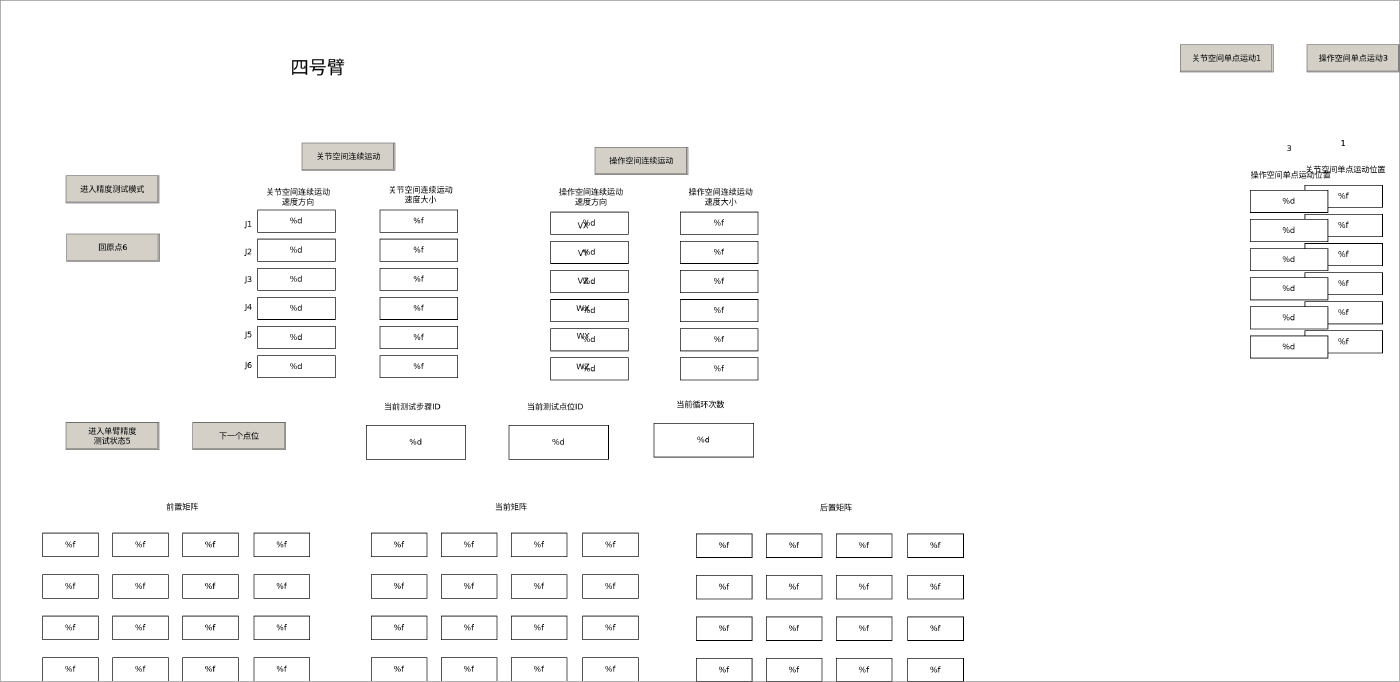
VISUALIZATION Robot_Jog_Arm4  // 1921x937
    Button (90,241 128x38), "进入精度测试模式", colour toggle: GVL_AccuracyTestVar.g_enterPrecisionTestMode[4]
        toggle GVL_AccuracyTestVar.g_enterPrecisionTestMode[4]
    Label (361,71 150x43), "四号臂"
    Group (1619,61 302x38), invisible if: TRUE
        Button (0,0 128x38), "关节空间单点运动1", colour toggle: A1_Arm1ModeL[4,1]
            tap A1_Arm1Mode[4,1]
        Button (174,0 128x38), "操作空间单点运动3", colour toggle: A1_Arm1ModeL[4,3]
            tap A1_Arm1Mode[4,3]
    Button (414,196 128x38), "关节空间连续运动", colour toggle: A1_Arm1ModeL[4,2]
        tap A1_Arm1Mode[4,2]
    Button (816,202 128x38), "操作空间连续运动", colour toggle: A1_Arm1ModeL[4,4]
        tap A1_Arm1Mode[4,4]
    Button (91,321 128x38), "回原点6", colour toggle: A1_Arm1ModeL[4,6]
        tap A1_Arm1Mode[4,6]
    Rectangle (353,288 107x31), "%d", text variable: GVL_AccuracyTestVar.g_jntMotionDir[4][1]
        OnMouseClick: write the text variable via Default, min -1, max 1
    Label (334,256 150x29), "关节空间连续运动 速度方向"
    Rectangle (353,328 107x31), "%d", text variable: GVL_AccuracyTestVar.g_jntMotionDir[4][2]
        OnMouseClick: write the text variable via Default, min -1, max 1
    Rectangle (353,368 107x31), "%d", text variable: GVL_AccuracyTestVar.g_jntMotionDir[4][3]
        OnMouseClick: write the text variable via Default, min -1, max 1
    Rectangle (353,408 107x31), "%d", text variable: GVL_AccuracyTestVar.g_jntMotionDir[4][4]
        OnMouseClick: write the text variable via Default, min -1, max 1
    Rectangle (353,448 107x31), "%d", text variable: GVL_AccuracyTestVar.g_jntMotionDir[4][5]
        OnMouseClick: write the text variable via Default, min -1, max 1
    Rectangle (353,488 107x31), "%d", text variable: GVL_AccuracyTestVar.g_jntMotionDir[4][6]
        OnMouseClick: write the text variable via Default, min -1, max 1
    Group (1768,182 153x303), invisible if: TRUE
        Rectangle (22,72 107x31), "%f", text variable: GVL_AccuracyTestVar.g_targetJntPos[4][1]
            OnMouseClick: write the text variable via Default
        Label (3,36 150x30), "关节空间单点运动位置"
        Rectangle (22,112 107x31), "%f", text variable: GVL_AccuracyTestVar.g_targetJntPos[4][2]
            OnMouseClick: write the text variable via Default
        Rectangle (22,152 107x31), "%f", text variable: GVL_AccuracyTestVar.g_targetJntPos[4][3]
            OnMouseClick: write the text variable via Default
        Rectangle (22,192 107x31), "%f", text variable: GVL_AccuracyTestVar.g_targetJntPos[4][4]
            OnMouseClick: write the text variable via Default
        Rectangle (22,232 107x31), "%f", text variable: GVL_AccuracyTestVar.g_targetJntPos[4][5]
            OnMouseClick: write the text variable via Default
        Rectangle (22,272 107x31), "%f", text variable: GVL_AccuracyTestVar.g_targetJntPos[4][6]
            OnMouseClick: write the text variable via Default
        Label (0,0 150x30), "1"
    Rectangle (521,288 107x31), "%f", text variable: GVL_AccuracyTestVar.g_jntVel[4][1]
        OnMouseClick: write the text variable via Default
    Label (502,253 150x29), "关节空间连续运动 速度大小"
    Rectangle (521,328 107x31), "%f", text variable: GVL_AccuracyTestVar.g_jntVel[4][2]
        OnMouseClick: write the text variable via Default
    Rectangle (521,368 107x31), "%f", text variable: GVL_AccuracyTestVar.g_jntVel[4][3]
        OnMouseClick: write the text variable via Default
    Rectangle (521,408 107x31), "%f", text variable: GVL_AccuracyTestVar.g_jntVel[4][4]
        OnMouseClick: write the text variable via Default
    Rectangle (521,448 107x31), "%f", text variable: GVL_AccuracyTestVar.g_jntVel[4][5]
        OnMouseClick: write the text variable via Default
    Rectangle (521,488 107x31), "%f", text variable: GVL_AccuracyTestVar.g_jntVel[4][6]
        OnMouseClick: write the text variable via Default
    Group (1694,189 152x303), invisible if: TRUE
        Rectangle (21,72 107x31), "%d"
        Label (2,37 150x29), "操作空间单点运动位置"
        Rectangle (21,112 107x31), "%d"
        Rectangle (21,152 107x31), "%d"
        Rectangle (21,192 107x31), "%d"
        Rectangle (21,232 107x31), "%d"
        Rectangle (21,272 107x31), "%d"
        Label (0,0 150x30), "3"
    Rectangle (755,291 107x31), "%d", text variable: GVL_AccuracyTestVar.g_spatialMotionDir[4][1]
        OnMouseClick: write the text variable via Default, min -1, max 1
    Label (736,256 150x29), "操作空间连续运动 速度方向"
    Rectangle (755,331 107x31), "%d", text variable: GVL_AccuracyTestVar.g_spatialMotionDir[4][2]
        OnMouseClick: write the text variable via Default, min -1, max 1
    Rectangle (755,371 107x31), "%d", text variable: GVL_AccuracyTestVar.g_spatialMotionDir[4][3]
        OnMouseClick: write the text variable via Default, min -1, max 1
    Rectangle (755,411 107x31), "%d", text variable: GVL_AccuracyTestVar.g_spatialMotionDir[4][4]
        OnMouseClick: write the text variable via Default, min -1, max 1
    Rectangle (755,451 107x31), "%d", text variable: GVL_AccuracyTestVar.g_spatialMotionDir[4][5]
        OnMouseClick: write the text variable via Default, min -1, max 1
    Rectangle (755,491 107x31), "%d", text variable: GVL_AccuracyTestVar.g_spatialMotionDir[4][6]
        OnMouseClick: write the text variable via Default, min -1, max 1
    Rectangle (933,291 107x31), "%f", text variable: GVL_AccuracyTestVar.g_spatialVel[4][1]
        OnMouseClick: write the text variable via Default
    Label (914,256 150x29), "操作空间连续运动 速度大小"
    Rectangle (933,331 107x31), "%f", text variable: GVL_AccuracyTestVar.g_spatialVel[4][2]
        OnMouseClick: write the text variable via Default
    Rectangle (933,371 107x31), "%f", text variable: GVL_AccuracyTestVar.g_spatialVel[4][3]
        OnMouseClick: write the text variable via Default
    Rectangle (933,411 107x31), "%f", text variable: GVL_AccuracyTestVar.g_spatialVel[4][4]
        OnMouseClick: write the text variable via Default
    Rectangle (933,451 107x31), "%f", text variable: GVL_AccuracyTestVar.g_spatialVel[4][5]
        OnMouseClick: write the text variable via Default
    Rectangle (933,491 107x31), "%f", text variable: GVL_AccuracyTestVar.g_spatialVel[4][6]
        OnMouseClick: write the text variable via Default
    Button (90,580 128x38), "进入单臂精度 测试状态5", colour toggle: A1_Arm1ModeL[4,5]
        tap A1_Arm1Mode[4,5]
    Button (264,580 128x38), "下一个点位", colour toggle: GVL_AccuracyTestVar.g_nextStep[4]
        tap GVL_AccuracyTestVar.g_nextStep[4]
    Group (491,541 545x90)
        Rectangle (11,43 137x47), "%d", text variable: GVL_AccuracyTestVar.g_curStep[4]
        Label (0,3 150x30), "当前测试步骤ID"
        Rectangle (207,43 137x47), "%d", text variable: GVL_AccuracyTestVar.g_testPointId[4]
        Label (196,3 150x30), "当前测试点位ID"
        Rectangle (406,40 137x47), "%d", text variable: GVL_AccuracyTestVar.g_testCycleId[4]
        Label (395,0 150x30), "当前循环次数"
    Group (334,293 14x224)
        Label (0,0 14x30), "J1"
        Label (0,38 14x30), "J2"
        Label (0,76 14x30), "J3"
        Label (0,114 14x30), "J4"
        Label (0,152 14x30), "J5"
        Label (0,194 14x30), "J6"
    Group (725,295 26x224)
        Label (0,0 150x30), "VX"
        Label (0,38 150x30), "VY"
        Label (0,76 150x30), "VZ"
        Label (0,114 150x30), "WX"
        Label (0,152 150x30), "WY"
        Label (0,194 150x30), "WZ"
    Label (175,682 150x29), "前置矩阵"
    Rectangle (58,732 77x33), "%f", text variable: GVL_AccuracyTestVar.g_frontPose[4].m_rot[1,1]
    Rectangle (154,732 77x33), "%f", text variable: GVL_AccuracyTestVar.g_frontPose[4].m_rot[1,2]
    Rectangle (250,732 77x33), "%f", text variable: GVL_AccuracyTestVar.g_frontPose[4].m_rot[1,3]
    Rectangle (348,732 77x33), "%f", text variable: GVL_AccuracyTestVar.g_frontPose[4].m_pos[1]
    Rectangle (58,789 77x33), "%f", text variable: GVL_AccuracyTestVar.g_frontPose[4].m_rot[2,1]
    Rectangle (58,846 77x33), "%f", text variable: GVL_AccuracyTestVar.g_frontPose[4].m_rot[3,1]
    Rectangle (58,903 77x33), "%f", text variable: 0
    Rectangle (154,789 77x33), "%f", text variable: GVL_AccuracyTestVar.g_frontPose[4].m_rot[2,2]
    Rectangle (250,789 77x33), "%f", text variable: GVL_AccuracyTestVar.g_frontPose[4].m_rot[2,3]
    Rectangle (348,789 77x33), "%f", text variable: GVL_AccuracyTestVar.g_frontPose[4].m_pos[2]
    Rectangle (154,846 77x33), "%f", text variable: GVL_AccuracyTestVar.g_frontPose[4].m_rot[3,2]
    Rectangle (250,846 77x33), "%f", text variable: GVL_AccuracyTestVar.g_frontPose[4].m_rot[3,3]
    Rectangle (348,846 77x33), "%f", text variable: GVL_AccuracyTestVar.g_frontPose[4].m_pos[3]
    Rectangle (154,903 77x33), "%f", text variable: 0
    Rectangle (250,903 77x33), "%f", text variable: 0
    Rectangle (348,903 77x33), "%f", text variable: 1
    Label (626,682 150x29), "当前矩阵"
    Rectangle (509,732 77x33), "%f", text variable: GVL_AccuracyTestVar.g_slaveArmPose[4].m_rot[1,1]
    Rectangle (605,732 77x33), "%f", text variable: GVL_AccuracyTestVar.g_slaveArmPose[4].m_rot[1,2]
    Rectangle (701,732 77x33), "%f", text variable: GVL_AccuracyTestVar.g_slaveArmPose[4].m_rot[1,3]
    Rectangle (799,732 77x33), "%f", text variable: GVL_AccuracyTestVar.g_slaveArmPose[4].m_pos[1]
    Rectangle (509,789 77x33), "%f", text variable: GVL_AccuracyTestVar.g_slaveArmPose[4].m_rot[2,1]
    Rectangle (509,846 77x33), "%f", text variable: GVL_AccuracyTestVar.g_slaveArmPose[4].m_rot[3,1]
    Rectangle (509,903 77x33), "%f", text variable: 0
    Rectangle (605,789 77x33), "%f", text variable: GVL_AccuracyTestVar.g_slaveArmPose[4].m_rot[2,2]
    Rectangle (701,789 77x33), "%f", text variable: GVL_AccuracyTestVar.g_slaveArmPose[4].m_rot[2,3]
    Rectangle (799,789 77x33), "%f", text variable: GVL_AccuracyTestVar.g_slaveArmPose[4].m_pos[2]
    Rectangle (605,846 77x33), "%f", text variable: GVL_AccuracyTestVar.g_slaveArmPose[4].m_rot[3,2]
    Rectangle (701,846 77x33), "%f", text variable: GVL_AccuracyTestVar.g_slaveArmPose[4].m_rot[3,3]
    Rectangle (799,846 77x33), "%f", text variable: GVL_AccuracyTestVar.g_slaveArmPose[4].m_pos[3]
    Rectangle (605,903 77x33), "%f", text variable: 0
    Rectangle (701,903 77x33), "%f", text variable: 0
    Rectangle (799,903 77x33), "%f", text variable: 1
    Label (1072,683 150x29), "后置矩阵"
    Rectangle (955,733 77x33), "%f", text variable: GVL_AccuracyTestVar.g_endPose[4].m_rot[1,1]
    Rectangle (1051,733 77x33), "%f", text variable: GVL_AccuracyTestVar.g_endPose[4].m_rot[1,2]
    Rectangle (1147,733 77x33), "%f", text variable: GVL_AccuracyTestVar.g_endPose[4].m_rot[1,3]
    Rectangle (1245,733 77x33), "%f", text variable: GVL_AccuracyTestVar.g_endPose[4].m_pos[1]
    Rectangle (955,790 77x33), "%f", text variable: GVL_AccuracyTestVar.g_endPose[4].m_rot[2,1]
    Rectangle (955,847 77x33), "%f", text variable: GVL_AccuracyTestVar.g_endPose[4].m_rot[3,1]
    Rectangle (955,904 77x33), "%f", text variable: 0
    Rectangle (1051,790 77x33), "%f", text variable: GVL_AccuracyTestVar.g_endPose[4].m_rot[2,2]
    Rectangle (1147,790 77x33), "%f", text variable: GVL_AccuracyTestVar.g_endPose[4].m_rot[2,3]
    Rectangle (1245,790 77x33), "%f", text variable: GVL_AccuracyTestVar.g_endPose[4].m_pos[2]
    Rectangle (1051,847 77x33), "%f", text variable: GVL_AccuracyTestVar.g_endPose[4].m_rot[3,2]
    Rectangle (1147,847 77x33), "%f", text variable: GVL_AccuracyTestVar.g_endPose[4].m_rot[3,3]
    Rectangle (1245,847 77x33), "%f", text variable: GVL_AccuracyTestVar.g_frontPose[4].m_pos[3]
    Rectangle (1051,904 77x33), "%f", text variable: 0
    Rectangle (1147,904 77x33), "%f", text variable: 0
    Rectangle (1245,904 77x33), "%f", text variable: 1
END_VISUALIZATION

(* stored: Version 1.1.0.1, ProductVersion 3.1.4024.11
   Visu Robot_Jog_Arm4: Id {aeaf9964-9823-479c-815c-e9ce5a32a76c} *)
